// TIA Portal project "sterowanieAnalogSilnikiem" (V15)

(* hardware
DEVICE "S7-1200 station_1"  S7-1200 Station
   slot 0: "Rack_0"  S7-1200 Rack  Rack  V1.0
   slot 1: "PLC_1"  CPU 1214C DC/DC/DC  6ES7 214-1AG40-0XB0  V4.2
      slot 3: "AQ 1x12BIT_1"  AQ1 signal board  6ES7 232-4HA30-0XB0  V1.0
   slot 101: "CM 1243-5"  CM 1243-5  6GK7 243-5DX30-0XE0  V1.3
   slot 102: "CM 1241 (RS485)_1"  CM 1241 (RS485)  6ES7 241-1CH30-0XB0  V1.0
*)

// ===== PLC "PLC_1"  CPU 1214C DC/DC/DC =====

VAR_GLOBAL   // PLC tag table "Default tag table"
   "Tag_1" AT %Q0.0 : Bool;
   "Tag_2" AT %M1.0 : Bool;
   "Tag_3" AT %M0.1 : Bool;
   "Tag_4" AT %M2.0 : Bool;
   "zalacz" AT %I0.7 : Bool;
   "Tag_7" AT %M3.0 : Bool;
   "zmniejszObrot" AT %I0.3 : Bool;
   "Tag_6" AT %M4.0 : Bool;
   "Tag_9" AT %QB0 : Byte;
   "Tag_10" AT %M5.0 : Bool;
   "Tag_11" AT %M0.0 : Bool;
   "Tag_12" AT %I0.0 : Bool;
   "Tag_13" AT %M10.0 : Bool;
   "Clock_Byte" AT %MB10 : Byte;
   "Clock_10Hz" AT %M10.0 : Bool;
   "Clock_5Hz" AT %M10.1 : Bool;
   "Clock_2.5Hz" AT %M10.2 : Bool;
   "Clock_2Hz" AT %M10.3 : Bool;
   "Clock_1.25Hz" AT %M10.4 : Bool;
   "Clock_1Hz" AT %M10.5 : Bool;
   "Clock_0.625Hz" AT %M10.6 : Bool;
   "Clock_0.5Hz" AT %M10.7 : Bool;
   "wartoscPotencjometru" AT %IW64 : Int;
   "Tag_15" AT %MD1000 : Real;
   "Tag_16" AT %MD1004 : Real;
   "Tag_17" AT %MW1008 : Int;
   "sterowanieSilnikiem" AT %QW80 : Int;
   "zalaczGenerator" AT %I0.6 : Bool;
   "sprzez" AT %M20.0 : Bool;
   "zwiekszObrot" AT %I0.2 : Bool;
   "predkoscObrotu" AT %MW80 : Word;
END_VAR

// folder: System blocks/Program resources

DATA_BLOCK "T1"   // DB1
{ S7_Optimized_Access := 'TRUE' }
AUTHOR : Simatic
FAMILY : IEC
NAME : IEC_TMR
VERSION : 1.0
// stored: InstanceOfName IEC_TIMER
"IEC_TIMER"
BEGIN
END_DATA_BLOCK

// folder: (top level)

FUNCTION "Block_1" : Void   // FC1, LAD
{ S7_Optimized_Access := 'TRUE' }
VERSION : 0.1
   VAR_INPUT
      potwierdzenie : Bool;
      gen : Bool;
      zaklocenie : Bool;
   END_VAR
   VAR_OUTPUT
      sygnal : Bool;
   END_VAR
   VAR_IN_OUT
      Pam_al_2 : Bool;
   END_VAR
   VAR_TEMP   // added for the SCL form of the ladder/FBD networks
      _w1 : Bool;
   END_VAR
BEGIN

REGION Network 1: Kanal Alarmowy
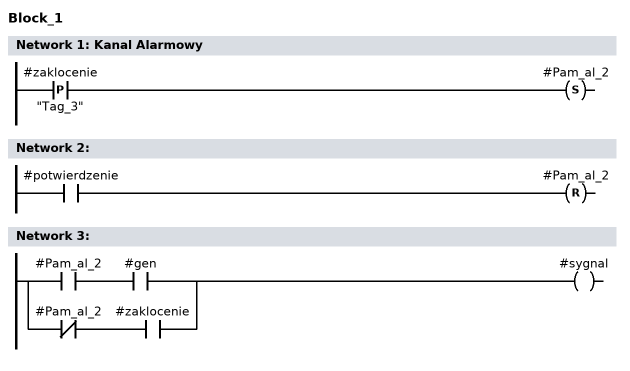
   RUNG wire#powerrail
      P_Contact(operand := #zaklocenie, bit := "Tag_3")
      S_Coil( #Pam_al_2 )
   END_RUNG
   // the same network as SCL:
   #_w1 := #zaklocenie AND NOT "Tag_3";   // rising edge of #zaklocenie
   "Tag_3" := #zaklocenie;
   IF #_w1 THEN #Pam_al_2 := TRUE; END_IF;
END_REGION

REGION Network 2
   RUNG wire#powerrail
      Contact( #potwierdzenie )
      R_Coil( #Pam_al_2 )
   END_RUNG
   // the same network as SCL:
   IF #potwierdzenie THEN #Pam_al_2 := FALSE; END_IF;
END_REGION

REGION Network 3
   RUNG wire#powerrail
      Contact( #Pam_al_2 )
      Contact( #gen )
      wire#w1
      Coil( #sygnal )
   END_RUNG
   RUNG wire#powerrail
      I_Contact( #Pam_al_2 )
      Contact( #zaklocenie )
   END_RUNG wire#w1
   // the same network as SCL:
   #sygnal := (#Pam_al_2 AND #gen) OR (NOT #Pam_al_2 AND #zaklocenie);
END_REGION
END_FUNCTION

ORGANIZATION_BLOCK "Main"   // OB1, LAD, ProgramCycle
TITLE = "Main Program Sweep (Cycle)"
{ S7_Optimized_Access := 'TRUE' }
VERSION : 0.1
   VAR_INPUT
      Initial_Call : Bool;   // Initial call of this OB
      Remanence : Bool;   // =True, if remanent data are available
   END_VAR
BEGIN

REGION Network 1: POTENCJOMETR
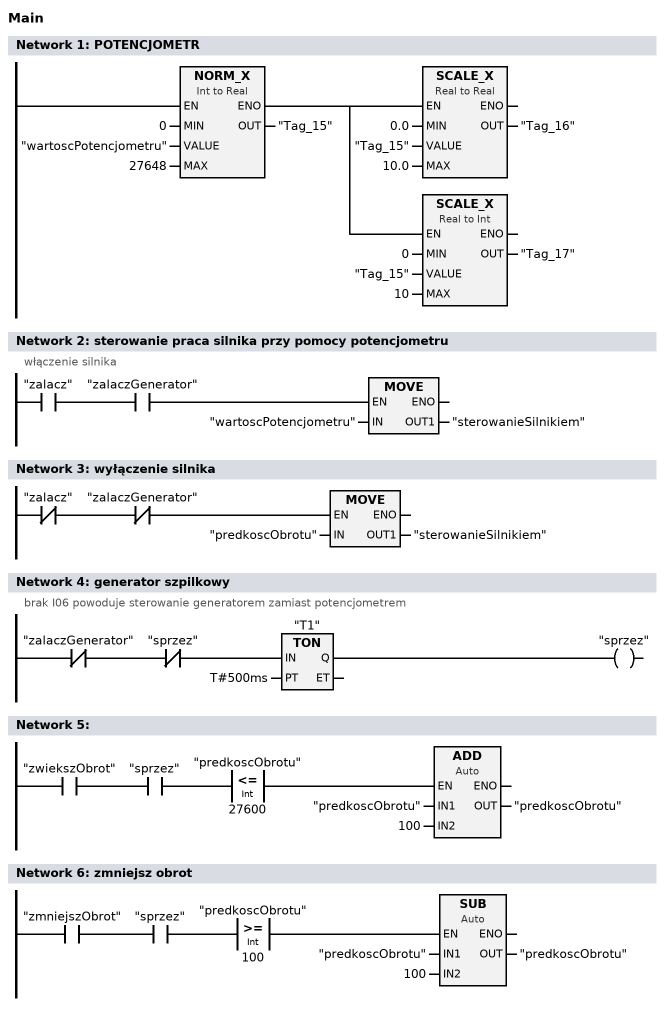
   RUNG wire#powerrail
      { S7_Templates := "[SrcType := Int, DestType := Real]" } Normalize(min := 0, value := "wartoscPotencjometru", max := 27648, out => "Tag_15")
      wire#w1
      { S7_Templates := "[SrcType := Real, DestType := Real]" } Scale(min := 0.0, value := "Tag_15", max := 10.0, out => "Tag_16")
   END_RUNG
   RUNG wire#w1
      { S7_Templates := "[SrcType := Real, DestType := Int]" } Scale(min := 0, value := "Tag_15", max := 10, out => "Tag_17")
   END_RUNG
   // the same network as SCL:
   "Tag_15" := NORM_X(MIN := 0, VALUE := "wartoscPotencjometru", MAX := 27648);
   "Tag_16" := SCALE_X(MIN := 0.0, VALUE := "Tag_15", MAX := 10.0);
   "Tag_17" := SCALE_X(MIN := 0, VALUE := "Tag_15", MAX := 10);
END_REGION

REGION Network 2: sterowanie praca silnika przy pomocy potencjometru
   // włączenie silnika
   RUNG wire#powerrail
      Contact( "zalacz" )
      Contact( "zalaczGenerator" )
      Move(in := "wartoscPotencjometru", out1 => "sterowanieSilnikiem")
   END_RUNG
   // the same network as SCL:
   IF "zalacz" AND "zalaczGenerator" THEN "sterowanieSilnikiem" := "wartoscPotencjometru"; END_IF;
END_REGION

REGION Network 3: wyłączenie silnika
   RUNG wire#powerrail
      I_Contact( "zalacz" )
      I_Contact( "zalaczGenerator" )
      Move(in := "predkoscObrotu", out1 => "sterowanieSilnikiem")
   END_RUNG
   // the same network as SCL:
   IF NOT "zalacz" AND NOT "zalaczGenerator" THEN "sterowanieSilnikiem" := "predkoscObrotu"; END_IF;
END_REGION

REGION Network 4: generator szpilkowy
   // brak I06 powoduje sterowanie generatorem zamiast potencjometrem
   "T1".TON(IN := NOT "zalaczGenerator" AND NOT "sprzez", PT := T#500ms);
   "sprzez" := "T1".Q;
END_REGION

REGION Network 5
   RUNG wire#powerrail
      Contact( "zwiekszObrot" )
      Contact( "sprzez" )
      { S7_Templates := "SrcType := Int" } LE_Contact(in1 := "predkoscObrotu", in2 := 27600)
      Add(in1 := "predkoscObrotu", in2 := 100, out => "predkoscObrotu")
   END_RUNG
   // the same network as SCL:
   IF "zwiekszObrot" AND "sprzez" AND ("predkoscObrotu" <= 27600) THEN
       "predkoscObrotu" := "predkoscObrotu" + 100;
   END_IF;
END_REGION

REGION Network 6: zmniejsz obrot
   RUNG wire#powerrail
      Contact( "zmniejszObrot" )
      Contact( "sprzez" )
      { S7_Templates := "SrcType := Int" } GE_Contact(in1 := "predkoscObrotu", in2 := 100)
      Sub(in1 := "predkoscObrotu", in2 := 100, out => "predkoscObrotu")
   END_RUNG
   // the same network as SCL:
   IF "zmniejszObrot" AND "sprzez" AND ("predkoscObrotu" >= 100) THEN
       "predkoscObrotu" := "predkoscObrotu" - 100;
   END_IF;
END_REGION
END_ORGANIZATION_BLOCK